Staubli VAL3: createtask.pgx

program createTask()
begin
  //Monitoring Task//
  taskCreate "MonitorTask",100,monitorTask()
  return
end
